TEXTLIST E_ParameterNames
  0 = 'Mpar_StitchLengthLong'
  1 = 'MPar_StitchLengthShort'
  2 = 'MPar_MaxSpeed'
  3 = 'Mpar_MinSpeed'
  4 = 'Mpar_ManualMaxSpeed'
  5 = 'Mpar_BacktackSpeed'
  6 = 'Mpar_SlowEndSpeed'
  7 = 'Mpar_HomingSpeed'
  8 = 'Mpar_CuttingSpeed'
  9 = 'Mpar_MaxAcceleration'
  10 = 'Mpar_MaxDeceleration'
  11 = 'Mpar_Jerk'
  12 = 'Mpar_BacktackAcceleration'
  13 = 'Mpar_BacktackDeceleration'
  14 = 'Mpar_TransferAcceleration'
  15 = 'Mpar_TransferDeceleration'
  16 = 'Mpar_CylinderTimeoutMargin'
  17 = 'Cpar_NeedleSensorPos'
  18 = 'Cpar_NeedlePosUp'
  19 = 'Cpar_NeedlePosInMaterial'
  20 = 'Cpar_NeedleposDown'
  21 = 'Cpar_NeedlePosStartCut'
  22 = 'Cpar_NeedlePosStopCut'
  23 = 'Cpar_NeedlePosEndCut'
  24 = 'Cpar_NeedlePosRelTensCut'
  25 = 'Cpar_NeedlePosHoldThread'
  26 = 'Cpar_NeedlePosStartRelTension'
  27 = 'Cpar_NeedlePosStopRelTension'
  28 = 'Cpar_NeedlePosChangeDirUp'
  29 = 'Cpar_NeedlePosClearStart'
  30 = 'Cpar_NeedlePosClearEnd'
  31 = 'Cpar_NeedlePosRef'
  32 = 'Cpar_NeedlePosPause'
  33 = 'Cpar_SensorPreEdgeDetDistance'
  34 = 'Cpar_sensorEdgeDetDistance'
  35 = 'Opar_NeedleSensorPos'
  36 = 'Opar_NeedlePosUp'
  37 = 'Opar_NeedlePosInMaterial'
  38 = 'Opar_NeedleposDown'
  39 = 'Opar_NeedlePosStartCut'
  40 = 'Opar_NeedlePosStopCut'
  41 = 'Opar_NeedlePosEndCut'
  42 = 'Opar_NeedlePosRelTensCut'
  43 = 'Opar_NeedlePosHoldThread'
  44 = 'Opar_NeedlePosStartRelTension'
  45 = 'Opar_NeedlePosStopRelTension'
  46 = 'Opar_NeedlePosChangeDir'
  47 = 'Opar_NeedlePosClearStart'
  48 = 'Opar_NeedlePosClearEnd'
  49 = 'Opar_NeedlePosPause'
  50 = 'Ppar_BacktackStitchStartFwd'
  51 = 'Ppar_BacktackStitchStartRev'
  52 = 'Ppar_BacktackStitchEndFwd'
  53 = 'Ppar_BacktackStitchEndRev'
  54 = 'Ppar_AutomaticSpeed'
  55 = 'Ppar_StitchStretch'
  56 = 'Ppar_ThreadLengthAdition'
  57 = 'Ppar_ThreadBreakDelay'
  58 = 'Mpar_MaxVelocity'
  59 = 'Mpar_MinVelocity'
  60 = 'Mpar_ManualMaxVelocity'
  61 = 'Mpar_MLTMaxAcceleration'
  62 = 'Mpar_MLTMaxDeceleration'
  63 = 'Mpar_TraverseLength'
  64 = 'Mpar_CylTimeOutMargine'
  65 = 'Mpar_HomingVelocity'
  66 = 'Mpar_SewingcartLength'
  67 = 'Mpar_ClampCartLength'
  68 = 'Mpar_MaxClampCartVelocity'
  69 = 'Mpar_TraverseReturnVelocity'
  70 = 'Mpar_ToStartvelocity'
  71 = 'Mpar_InspectionDistance'
  72 = 'Cpar_PosHoming'
  73 = 'Cpar_PosSuportCyl_1'
  74 = 'Cpar_PosSuportCyl_2'
  75 = 'Cpar_PosSuportCyl_3'
  76 = 'Cpar_PosService'
  77 = 'Cpar_PosBobinChange'
  78 = 'Cpar_PosEnd'
  79 = 'Cpar_TimeBaseClampsClose'
  80 = 'Cpar_TimeBaseClampsRel'
  81 = 'Cpar_TimeCartClampsClose'
  82 = 'Cpar_TimeCartClampsRel'
  83 = 'Cpar_TimeCartBrakeApply'
  84 = 'Cpar_TimeCartBrakeRel'
  85 = 'Cpar_TimeSupportExp_1'
  86 = 'Cpar_TimeSupportRet_1'
  87 = 'Cpar_TimeSupportExp_2'
  88 = 'Cpar_TimeSupportRet_2'
  89 = 'Cpar_TimeSupportExp_3'
  90 = 'Cpar_TimeSupportRet_3'
  91 = 'Cpar_TimeBobinPlateClose'
  92 = 'Cpar_TimeBobinPlateOpen'
  93 = 'Cpar_PosFlagSewingcart'
  94 = 'Cpar_PosSensorClampCart'
  95 = 'Cpar_SupportCylWidth'
  96 = 'Cpar_ClampCartFlagWidth'
  97 = 'Cpar_PosMaterialStart'
  98 = 'Opar_HomePosition'
  99 = 'Opar_PosSuportCyl_1'
  100 = 'Opar_PosSuportCyl_2'
  101 = 'Opar_PosSuportCyl_3'
  102 = 'Opar_PosService'
  103 = 'Opar_PosBobinChange'
  104 = 'Opar_PosEnd'
  105 = 'Opar_PosMatStart'
  106 = 'Ppar_ProductLenght'
  107 = 'Ppar_ProductStretch'
  108 = 'Ppar_StartStretchFactor'
  109 = 'Ppar_StartStretchLength'
  110 = 'Ppar_ReverseStretch'
  111 = 'Ppar_MatBlowDistance'
   = ''
END_TEXTLIST

(* stored: Version 1.1.0.1, ProductVersion 3.1.4024.3
   TextList E_ParameterNames: Id {40009220-a4d3-4ff1-8d80-2968c0d6ce99} *)
